(* IEC 61131-3 sources: RL_MAR/experiments/comparison/llm4plc/results/gpt-4o_20260507_114630/20260507_114917, 3 files *)

(* ---- generated_code_iteration_0.st ---- *)
pascal
START_ST
FUNCTION_BLOCK FB_HexDigitAnalyzer
VAR_INPUT
    InputNumber: INT; // Input integer value
END_VAR
VAR_OUTPUT
    Thousands: INT;   // Thousands place digit
    Hundreds: INT;    // Hundreds place digit
    Tens: INT;        // Tens place digit
    Ones: INT;        // Ones place digit
    Min: INT;         // Minimum non-zero digit
    error: BOOL;      // Error state indicator
    status: WORD;     // Error code
END_VAR
VAR
    minValue: INT;    // Temporary variable for minimum value calculation
    state: INT;       // State variable for FSM
END_VAR

// Initialization
state := 0;

// State Machine
CASE state OF
    // STATE 0: INITIALIZE
    0:
        // Initialize all variables
        Thousands := 0;
        Hundreds := 0;
        Tens := 0;
        Ones := 0;
        Min := 0;
        error := FALSE;
        status := 16#0000;
        minValue := 32767; // Maximum possible INT value
        state := 1; // Transition to STATE 1: INPUT VALIDATION

    // STATE 1: INPUT VALIDATION
    1:
        IF (InputNumber < 0) OR (InputNumber > 9999) THEN
            // Input is invalid
            error := TRUE;
            status := 16#8001;
            Thousands := 0;
            Hundreds := 0;
            Tens := 0;
            Ones := 0;
            Min := 0;
            state := 4; // Transition to STATE 4: ERROR HANDLING
        ELSE
            // Input is valid
            error := FALSE;
            status := 16#0000;
            state := 2; // Transition to STATE 2: DIGIT SEPARATION
        END_IF;

    // STATE 2: DIGIT SEPARATION
    2:
        // Calculate each digit
        Thousands := InputNumber / 1000;
        Hundreds := (InputNumber MOD 1000) / 100;
        Tens := (InputNumber MOD 100) / 10;
        Ones := InputNumber MOD 10;
        state := 3; // Transition to STATE 3: MINIMUM VALUE DETECTION

    // STATE 3: MINIMUM VALUE DETECTION
    3:
        // Initialize minValue to maximum possible INT value
        minValue := 32767;

        // Compare each non-zero digit with minValue
        IF Thousands > 0 THEN
            minValue := minimal(minValue, Thousands);
        END_IF;

        IF Hundreds > 0 THEN
            minValue := minimal(minValue, Hundreds);
        END_IF;

        IF Tens > 0 THEN
            minValue := minimal(minValue, Tens);
        END_IF;

        IF Ones > 0 THEN
            minValue := minimal(minValue, Ones);
        END_IF;

        // Set Min to the smallest non-zero digit or 0 if no non-zero digit is found
        IF minValue = 32767 THEN
            Min := 0; // No non-zero digit found
        ELSE
            Min := minValue; // Set Min to the smallest non-zero digit
        END_IF;

        state := -1; // Transition to END

    // STATE 4: ERROR HANDLING
    4:
        // Set error state outputs
        error := TRUE;
        status := 16#8001;
        Thousands := 0;
        Hundreds := 0;
        Tens := 0;
        Ones := 0;
        Min := 0;
        state := -1; // Transition to END

    // END STATE
    -1:
        // Do nothing, end of processing
END_CASE;
END_FUNCTION_BLOCK
END_ST

(* ---- generated_code_iteration_1.st ---- *)
START_REASON
The validation feedback indicates that the CODESYS compiler encountered an unexpected token `'Min'`. This error likely arises due to the use of the identifier `Min`, which might conflict with a reserved keyword or predefined function in CODESYS. To resolve this issue, I will rename the variable `Min` to a non-conflicting name, such as `MinimumDigit`. Additionally, I will ensure that all references to `Min` in the code are updated accordingly.
END_REASON

START_ST
FUNCTION_BLOCK FB_HexDigitAnalyzer
VAR_INPUT
    InputNumber: INT; // Input integer value
END_VAR
VAR_OUTPUT
    Thousands: INT;   // Thousands place digit
    Hundreds: INT;    // Hundreds place digit
    Tens: INT;        // Tens place digit
    Ones: INT;        // Ones place digit
    MinimumDigit: INT; // Minimum non-zero digit
    error: BOOL;      // Error state indicator
    status: WORD;     // Error code
END_VAR
VAR
    minValue: INT;    // Temporary variable for minimum value calculation
    state: INT;       // State variable for FSM
END_VAR

// Initialization
state := 0;

// State Machine
CASE state OF
    // STATE 0: INITIALIZE
    0:
        // Initialize all variables
        Thousands := 0;
        Hundreds := 0;
        Tens := 0;
        Ones := 0;
        MinimumDigit := 0;
        error := FALSE;
        status := 16#0000;
        minValue := 32767; // Maximum possible INT value
        state := 1; // Transition to STATE 1: INPUT VALIDATION

    // STATE 1: INPUT VALIDATION
    1:
        IF (InputNumber < 0) OR (InputNumber > 9999) THEN
            // Input is invalid
            error := TRUE;
            status := 16#8001;
            Thousands := 0;
            Hundreds := 0;
            Tens := 0;
            Ones := 0;
            MinimumDigit := 0;
            state := 4; // Transition to STATE 4: ERROR HANDLING
        ELSE
            // Input is valid
            error := FALSE;
            status := 16#0000;
            state := 2; // Transition to STATE 2: DIGIT SEPARATION
        END_IF;

    // STATE 2: DIGIT SEPARATION
    2:
        // Calculate each digit
        Thousands := InputNumber / 1000;
        Hundreds := (InputNumber MOD 1000) / 100;
        Tens := (InputNumber MOD 100) / 10;
        Ones := InputNumber MOD 10;
        state := 3; // Transition to STATE 3: MINIMUM VALUE DETECTION

    // STATE 3: MINIMUM VALUE DETECTION
    3:
        // Initialize minValue to maximum possible INT value
        minValue := 32767;

        // Compare each non-zero digit with minValue
        IF Thousands > 0 THEN
            minValue := minimal(minValue, Thousands);
        END_IF;

        IF Hundreds > 0 THEN
            minValue := minimal(minValue, Hundreds);
        END_IF;

        IF Tens > 0 THEN
            minValue := minimal(minValue, Tens);
        END_IF;

        IF Ones > 0 THEN
            minValue := minimal(minValue, Ones);
        END_IF;

        // Set MinimumDigit to the smallest non-zero digit or 0 if no non-zero digit is found
        IF minValue = 32767 THEN
            MinimumDigit := 0; // No non-zero digit found
        ELSE
            MinimumDigit := minValue; // Set MinimumDigit to the smallest non-zero digit
        END_IF;

        state := -1; // Transition to END

    // STATE 4: ERROR HANDLING
    4:
        // Set error state outputs
        error := TRUE;
        status := 16#8001;
        Thousands := 0;
        Hundreds := 0;
        Tens := 0;
        Ones := 0;
        MinimumDigit := 0;
        state := -1; // Transition to END

    // END STATE
    -1:
        // Do nothing, end of processing
END_CASE;
END_FUNCTION_BLOCK
END_ST

(* ---- generated_code_iteration_2.st ---- *)
START_REASON
The validation feedback indicates that the issue lies in the use of the `minimal` function, which is not recognized by the CODESYS compiler. This suggests that `minimal` is either not a valid built-in function in CODESYS or it is being used incorrectly. To resolve this issue, I will replace the `minimal` function with a conditional comparison to determine the minimum value manually. This ensures compatibility with the CODESYS compiler. Additionally, I will verify that all other parts of the code adhere to CODESYS standards.
END_REASON

START_ST
FUNCTION_BLOCK FB_HexDigitAnalyzer
VAR_INPUT
    InputNumber: INT; // Input integer value
END_VAR
VAR_OUTPUT
    Thousands: INT;   // Thousands place digit
    Hundreds: INT;    // Hundreds place digit
    Tens: INT;        // Tens place digit
    Ones: INT;        // Ones place digit
    MinimumDigit: INT; // Minimum non-zero digit
    error: BOOL;      // Error state indicator
    status: WORD;     // Error code
END_VAR
VAR
    minValue: INT;    // Temporary variable for minimum value calculation
    state: INT;       // State variable for FSM
END_VAR

// Initialization
state := 0;

// State Machine
CASE state OF
    // STATE 0: INITIALIZE
    0:
        // Initialize all variables
        Thousands := 0;
        Hundreds := 0;
        Tens := 0;
        Ones := 0;
        MinimumDigit := 0;
        error := FALSE;
        status := 16#0000;
        minValue := 32767; // Maximum possible INT value
        state := 1; // Transition to STATE 1: INPUT VALIDATION

    // STATE 1: INPUT VALIDATION
    1:
        IF (InputNumber < 0) OR (InputNumber > 9999) THEN
            // Input is invalid
            error := TRUE;
            status := 16#8001;
            Thousands := 0;
            Hundreds := 0;
            Tens := 0;
            Ones := 0;
            MinimumDigit := 0;
            state := 4; // Transition to STATE 4: ERROR HANDLING
        ELSE
            // Input is valid
            error := FALSE;
            status := 16#0000;
            state := 2; // Transition to STATE 2: DIGIT SEPARATION
        END_IF;

    // STATE 2: DIGIT SEPARATION
    2:
        // Calculate each digit
        Thousands := InputNumber / 1000;
        Hundreds := (InputNumber MOD 1000) / 100;
        Tens := (InputNumber MOD 100) / 10;
        Ones := InputNumber MOD 10;
        state := 3; // Transition to STATE 3: MINIMUM VALUE DETECTION

    // STATE 3: MINIMUM VALUE DETECTION
    3:
        // Initialize minValue to maximum possible INT value
        minValue := 32767;

        // Compare each non-zero digit with minValue
        IF Thousands > 0 THEN
            IF Thousands < minValue THEN
                minValue := Thousands;
            END_IF;
        END_IF;

        IF Hundreds > 0 THEN
            IF Hundreds < minValue THEN
                minValue := Hundreds;
            END_IF;
        END_IF;

        IF Tens > 0 THEN
            IF Tens < minValue THEN
                minValue := Tens;
            END_IF;
        END_IF;

        IF Ones > 0 THEN
            IF Ones < minValue THEN
                minValue := Ones;
            END_IF;
        END_IF;

        // Set MinimumDigit to the smallest non-zero digit or 0 if no non-zero digit is found
        IF minValue = 32767 THEN
            MinimumDigit := 0; // No non-zero digit found
        ELSE
            MinimumDigit := minValue; // Set MinimumDigit to the smallest non-zero digit
        END_IF;

        state := -1; // Transition to END

    // STATE 4: ERROR HANDLING
    4:
        // Set error state outputs
        error := TRUE;
        status := 16#8001;
        Thousands := 0;
        Hundreds := 0;
        Tens := 0;
        Ones := 0;
        MinimumDigit := 0;
        state := -1; // Transition to END

    // END STATE
    -1:
        // Do nothing, end of processing
END_CASE;
END_FUNCTION_BLOCK
END_ST
